PROGRAM PRG_TEST
VAR
	fb_GeoPosition : FB_GeoPosition_Test;
	fb_GeoEllipsoid : FB_GeoEllipsoid_Test;
END_VAR

TcUnit.RUN();

END_PROGRAM

(* stored: Version 1.1.0.1, ProductVersion 3.1.4024.9
   POU PRG_TEST: Id {f534f62b-6a4d-4076-89d7-d888d6ef7143}, SpecialFunc None *)
